FUNCTION_BLOCK LED_Controller (* Composite Function Block Type *)
  (* Standard: 61499-2 *)
  (* Version 0.0, 9/22/2026, macie, Schneider Electric, template *)
  PACKAGE Main;
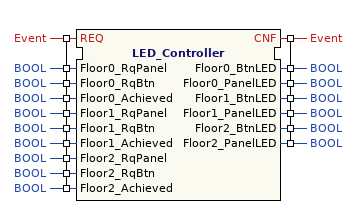
  EVENT_INPUT
    REQ WITH Floor0_RqPanel, Floor0_RqBtn, Floor0_Achieved, Floor1_RqPanel, Floor1_RqBtn, Floor1_Achieved, Floor2_RqPanel, Floor2_RqBtn, Floor2_Achieved; (* Normal Execution Request *)
  END_EVENT
  EVENT_OUTPUT
    CNF WITH Floor0_BtnLED, Floor0_PanelLED, Floor1_BtnLED, Floor1_PanelLED, Floor2_BtnLED, Floor2_PanelLED; (* Execution Confirmation *)
  END_EVENT
  VAR_INPUT
    Floor0_RqPanel : BOOL; (* Input event qualifier *)
    Floor0_RqBtn : BOOL;
    Floor0_Achieved : BOOL;
    Floor1_RqPanel : BOOL;
    Floor1_RqBtn : BOOL;
    Floor1_Achieved : BOOL;
    Floor2_RqPanel : BOOL;
    Floor2_RqBtn : BOOL;
    Floor2_Achieved : BOOL;
  END_VAR
  VAR_OUTPUT
    Floor0_BtnLED : BOOL := FALSE; (* Output event qualifier *)
    Floor0_PanelLED : BOOL := FALSE;
    Floor1_BtnLED : BOOL := FALSE;
    Floor1_PanelLED : BOOL := FALSE;
    Floor2_BtnLED : BOOL := FALSE;
    Floor2_PanelLED : BOOL := FALSE;
  END_VAR
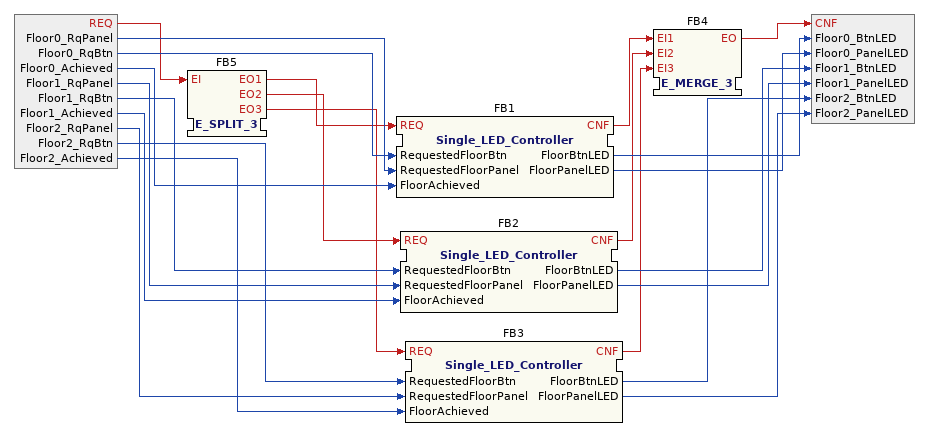
  FBS
    FB1 : Single_LED_Controller;
    FB2 : Single_LED_Controller;
    FB3 : Single_LED_Controller;
    FB4 : E_MERGE_3;
    FB5 : E_SPLIT_3;
  END_FBS
  EVENT_CONNECTIONS
    FB2.CNF TO FB4.EI2;
    FB1.CNF TO FB4.EI1;
    FB3.CNF TO FB4.EI3;
    FB4.EO TO CNF;
    REQ TO FB5.EI;
    FB5.EO1 TO FB1.REQ;
    FB5.EO2 TO FB2.REQ;
    FB5.EO3 TO FB3.REQ;
  END_CONNECTIONS
  DATA_CONNECTIONS
    FB1.FloorBtnLED TO Floor0_BtnLED;
    FB2.FloorBtnLED TO Floor1_BtnLED;
    FB3.FloorBtnLED TO Floor2_BtnLED;
    Floor0_RqPanel TO FB1.RequestedFloorPanel;
    Floor0_Achieved TO FB1.FloorAchieved;
    Floor1_RqPanel TO FB2.RequestedFloorPanel;
    Floor1_Achieved TO FB2.FloorAchieved;
    Floor2_Achieved TO FB3.FloorAchieved;
    Floor2_RqPanel TO FB3.RequestedFloorPanel;
    Floor0_RqBtn TO FB1.RequestedFloorBtn;
    Floor1_RqBtn TO FB2.RequestedFloorBtn;
    Floor2_RqBtn TO FB3.RequestedFloorBtn;
    FB3.FloorPanelLED TO Floor2_PanelLED;
    FB2.FloorPanelLED TO Floor1_PanelLED;
    FB1.FloorPanelLED TO Floor0_PanelLED;
  END_CONNECTIONS
END_FUNCTION_BLOCK
